(* IEC 61131-3 sources: lacyccom/src/Types/serde, 6 files *)

(* ---- LAcycCom_Typestatheader.st ---- *)
// This is generated code. *** DO NOT MODIFY ***

NAMESPACE Simatic.Ax.LAcycCom
FUNCTION SerializeBig : UINT
    VAR_INPUT
        offset : UINT;
        value : LAcycCom_Typestatheader;
    END_VAR
    VAR_IN_OUT
        buffer : ARRAY[*] OF BYTE;
    END_VAR
    SerializeBig := offset;
    SerializeBig := System.Serde.SerializeBig(offset := SerializeBig, value := value.refNo, buffer := buffer);
    SerializeBig := System.Serde.SerializeBig(offset := SerializeBig, value := value.reqId, buffer := buffer);
    SerializeBig := System.Serde.SerializeBig(offset := SerializeBig, value := value.doId, buffer := buffer);
    SerializeBig := System.Serde.SerializeBig(offset := SerializeBig, value := value.parameterNo, buffer := buffer);
END_FUNCTION

FUNCTION DeserializeBig : UINT
    VAR_INPUT
        offset : UINT;
        buffer : ARRAY[*] OF BYTE;
    END_VAR
    VAR_IN_OUT
        value : LAcycCom_Typestatheader;
    END_VAR
    DeserializeBig := offset;
    DeserializeBig := System.Serde.DeserializeBig(offset := DeserializeBig, value := value.refNo, buffer := buffer);
    DeserializeBig := System.Serde.DeserializeBig(offset := DeserializeBig, value := value.reqId, buffer := buffer);
    DeserializeBig := System.Serde.DeserializeBig(offset := DeserializeBig, value := value.doId, buffer := buffer);
    DeserializeBig := System.Serde.DeserializeBig(offset := DeserializeBig, value := value.parameterNo, buffer := buffer);
END_FUNCTION
END_NAMESPACE

(* ---- LAcycCom_TypestatparameterAddress.st ---- *)
// This is generated code. *** DO NOT MODIFY ***

NAMESPACE Simatic.Ax.LAcycCom
FUNCTION SerializeBig : UDINT
    VAR_INPUT
        offset : UDINT;
        value : LAcycCom_TypestatparameterAddress;
    END_VAR
    VAR_IN_OUT
        buffer : ARRAY[*] OF BYTE;
    END_VAR
    SerializeBig := offset;
    SerializeBig := System.Serialization.SerializeBig(offset := SerializeBig, value := value.attribute, buffer := buffer);
    SerializeBig := System.Serialization.SerializeBig(offset := SerializeBig, value := value.elementNo, buffer := buffer);
    SerializeBig := System.Serialization.SerializeBig(offset := SerializeBig, value := value.parameterNo, buffer := buffer);
    SerializeBig := System.Serialization.SerializeBig(offset := SerializeBig, value := value.index, buffer := buffer);
END_FUNCTION

FUNCTION DeserializeBig : UDINT
    VAR_INPUT
        offset : UDINT;
        buffer : ARRAY[*] OF BYTE;
    END_VAR
    VAR_IN_OUT
        value : LAcycCom_TypestatparameterAddress;
    END_VAR
    DeserializeBig := offset;
    DeserializeBig := System.Serialization.DeserializeBig(offset := DeserializeBig, value := value.attribute, buffer := buffer);
    DeserializeBig := System.Serialization.DeserializeBig(offset := DeserializeBig, value := value.elementNo, buffer := buffer);
    DeserializeBig := System.Serialization.DeserializeBig(offset := DeserializeBig, value := value.parameterNo, buffer := buffer);
    DeserializeBig := System.Serialization.DeserializeBig(offset := DeserializeBig, value := value.index, buffer := buffer);
END_FUNCTION
END_NAMESPACE

(* ---- LAcycCom_TypestatReqReadParameter.st ---- *)
// This is generated code. *** DO NOT MODIFY ***

NAMESPACE Simatic.Ax.LAcycCom
FUNCTION SerializeBig : UDINT
    VAR_INPUT
        offset : UDINT;
        value : LAcycCom_TypestatReqReadParameter;
    END_VAR
    VAR_IN_OUT
        buffer : ARRAY[*] OF BYTE;
    END_VAR
    VAR_TEMP
        i : INT;
    END_VAR
    SerializeBig := offset;
    SerializeBig := LAcycCom.SerializeBig(offset := SerializeBig, value := value.header, buffer := buffer);
    FOR i := 0 TO 0 DO
        SerializeBig := LAcycCom.SerializeBig(offset := SerializeBig, value := value.parameterAddress[i], buffer := buffer);
    END_FOR;
END_FUNCTION

FUNCTION DeserializeBig : UDINT
    VAR_INPUT
        offset : UDINT;
        buffer : ARRAY[*] OF BYTE;
    END_VAR
    VAR_IN_OUT
        value : LAcycCom_TypestatReqReadParameter;
    END_VAR
    VAR_TEMP
        i : INT;
    END_VAR
    DeserializeBig := offset;
    DeserializeBig := LAcycCom.DeserializeBig(offset := DeserializeBig, value := value.header, buffer := buffer);
    FOR i := 0 TO 0 DO
        DeserializeBig := LAcycCom.DeserializeBig(offset := DeserializeBig, value := value.parameterAddress[i], buffer := buffer);
    END_FOR;
END_FUNCTION
END_NAMESPACE

(* ---- LAcycCom_TypestatReqWriteParameter.st ---- *)
// This is generated code. *** DO NOT MODIFY ***

NAMESPACE Simatic.Ax.LAcycCom
FUNCTION SerializeBig : UDINT
    VAR_INPUT
        offset : UDINT;
        value : LAcycCom_TypestatReqWriteParameter;
    END_VAR
    VAR_IN_OUT
        buffer : ARRAY[*] OF BYTE;
    END_VAR
    VAR_TEMP
        i : INT;
    END_VAR
    SerializeBig := offset;
    SerializeBig := LAcycCom.SerializeBig(offset := SerializeBig, value := value.header, buffer := buffer);
    FOR i := 0 TO 227 DO
        SerializeBig := System.Serialization.SerializeBig(offset := SerializeBig, value := value.data[i], buffer := buffer);
    END_FOR;
END_FUNCTION

FUNCTION DeserializeBig : UDINT
    VAR_INPUT
        offset : UDINT;
        buffer : ARRAY[*] OF BYTE;
    END_VAR
    VAR_IN_OUT
        value : LAcycCom_TypestatReqWriteParameter;
    END_VAR
    VAR_TEMP
        i : INT;
    END_VAR
    DeserializeBig := offset;
    DeserializeBig := LAcycCom.DeserializeBig(offset := DeserializeBig, value := value.header, buffer := buffer);
    FOR i := 0 TO 227 DO
        DeserializeBig := System.Serialization.DeserializeBig(offset := DeserializeBig, value := value.data[i], buffer := buffer);
    END_FOR;
END_FUNCTION
END_NAMESPACE

(* ---- LAcycCom_TypestatRespParameter.st ---- *)
// This is generated code. *** DO NOT MODIFY ***

NAMESPACE Simatic.Ax.LAcycCom
FUNCTION SerializeBig : UDINT
    VAR_INPUT
        offset : UDINT;
        value : LAcycCom_TypestatRespParameter;
    END_VAR
    VAR_IN_OUT
        buffer : ARRAY[*] OF BYTE;
    END_VAR
    VAR_TEMP
        i : INT;
    END_VAR
    SerializeBig := offset;
    SerializeBig := LAcycCom.SerializeBig(offset := SerializeBig, value := value.header, buffer := buffer);
    FOR i := 0 TO 233 DO
        SerializeBig := System.Serialization.SerializeBig(offset := SerializeBig, value := value.data[i], buffer := buffer);
    END_FOR;
END_FUNCTION

FUNCTION DeserializeBig : UDINT
    VAR_INPUT
        offset : UDINT;
        buffer : ARRAY[*] OF BYTE;
    END_VAR
    VAR_IN_OUT
        value : LAcycCom_TypestatRespParameter;
    END_VAR
    VAR_TEMP
        i : INT;
    END_VAR
    DeserializeBig := offset;
    DeserializeBig := LAcycCom.DeserializeBig(offset := DeserializeBig, value := value.header, buffer := buffer);
    FOR i := 0 TO 233 DO
        DeserializeBig := System.Serialization.DeserializeBig(offset := DeserializeBig, value := value.data[i], buffer := buffer);
    END_FOR;
END_FUNCTION
END_NAMESPACE

(* ---- LAcycCom_TypestatstatReqParameter.st ---- *)
// This is generated code. *** DO NOT MODIFY ***

NAMESPACE Simatic.Ax.LAcycCom
FUNCTION SerializeBig : UDINT
    VAR_INPUT
        offset : UDINT;
        value : LAcycCom_TypestatstatReqParameter;
    END_VAR
    VAR_IN_OUT
        buffer : ARRAY[*] OF BYTE;
    END_VAR
    VAR_TEMP
        i : INT;
    END_VAR
    SerializeBig := offset;
    SerializeBig := LAcycCom.SerializeBig(offset := SerializeBig, value := value.header, buffer := buffer);
    FOR i := 0 TO 38 DO
        SerializeBig := LAcycCom.SerializeBig(offset := SerializeBig, value := value.parameterAddress[i], buffer := buffer);
    END_FOR;
END_FUNCTION

FUNCTION DeserializeBig : UDINT
    VAR_INPUT
        offset : UDINT;
        buffer : ARRAY[*] OF BYTE;
    END_VAR
    VAR_IN_OUT
        value : LAcycCom_TypestatstatReqParameter;
    END_VAR
    VAR_TEMP
        i : INT;
    END_VAR
    DeserializeBig := offset;
    DeserializeBig := LAcycCom.DeserializeBig(offset := DeserializeBig, value := value.header, buffer := buffer);
    FOR i := 0 TO 38 DO
        DeserializeBig := LAcycCom.DeserializeBig(offset := DeserializeBig, value := value.parameterAddress[i], buffer := buffer);
    END_FOR;
END_FUNCTION
END_NAMESPACE
